{attribute 'linkalways'} 
{attribute 'no_explicit_call' := 'This FB is a CLASS and must be accessed using methods or properties'}
{attribute 'enable_dynamic_creation'}
FUNCTION_BLOCK Node_F_VN_CreateHighpassButterworthFilter EXTENDS VisionNode
VAR
    ipFilter : _ITcVnImage;
    nWidth : _UDINT(2);
    nHeight : _UDINT(2);
    bDoublePrecision : _BOOL(FALSE);
    bOriginAtCenter : _BOOL(FALSE);
    fCutoffDistance : _LREAL(1.0);
    nOrder : _UDINT(1);
    fScale : _LREAL(1.0);
    hrPrev : _HRESULT(S_OK);
	hresult : _HRESULT(S_OK);
END_VAR

METHOD PUBLIC  Clone : I_Node
VAR
	pNode : POINTER TO Node_F_VN_CreateHighpassButterworthFilter;
END_VAR
pNode := __NEW(Node_F_VN_CreateHighpassButterworthFilter);
Clone := pNode^;
END_METHOD

METHOD FB_init : BOOL
VAR_INPUT
	bInitRetains : BOOL; // if TRUE, the retain variables are initialized (warm start / cold start)
	bInCopyCode : BOOL;  // if TRUE, the instance afterwards gets moved into the copy code (online change)
END_VAR
AddParameter('nWidth', nWidth);
AddParameter('nHeight', nHeight);
AddParameter('bDoublePrecision', bDoublePrecision);
AddParameter('bOriginAtCenter', bOriginAtCenter);
AddParameter('fCutoffDistance', fCutoffDistance);
AddParameter('nOrder', nOrder);
AddParameter('fScale', fScale);
AddInput('hrPrev', hrPrev);
AddOutput('ipFilter', ipFilter);
AddOutput('hresult',hresult);
END_METHOD

METHOD PROTECTED OnExecute
hresult.Value := F_VN_CreateHighpassButterworthFilter(
    ipFilter := ipFilter.Value,
	nWidth := nWidth.Value,
    nHeight := nHeight.Value,
    bDoublePrecision := bDoublePrecision.Value,
    bOriginAtCenter := bOriginAtCenter.Value,
    fCutoffDistance := fCutoffDistance.Value,
    nOrder := nOrder.Value,
    fScale := fScale.Value,
	hrPrev:= hrPrev.Value);
END_METHOD

METHOD PUBLIC PreExecutionCheck
VAR_INPUT
	Check : I_PreExecutionChecks;
END_VAR
Check.IsTrue(nWidth.IsEven, 'nWidth must be an even number');
Check.IsTrue(nHeight.IsEven, 'nHeight must be an even number');
Check.IsTrue((nWidth.Value >= 2), 'nWidth must be greater than or equal to 2');
Check.IsTrue((nHeight.Value >= 2), 'nWidth must be greater than or equal to 2');
Check.IsTrue((fCutoffDistance.Value > 0), 'nCutoffDistance must be greater than 0');
Check.IsTrue((nOrder.Value > 0), 'nOrder must be greater than 0');
Check.IsTrue((fScale.Value > 0), 'fScale must be greater than 0');
END_METHOD

END_FUNCTION_BLOCK

(* stored: Version 1.1.0.1, ProductVersion 3.1.4024.13
   POU Node_F_VN_CreateHighpassButterworthFilter: Id {e6d8493b-b689-0c34-30ba-ecc7acc460ab}, SpecialFunc None
   Folder Constructor: Id {10b100ae-515d-058b-0a31-404109c7c72b}
   Method Clone: Id {01652cac-4fbc-0893-23d7-e4b31a061049}
   Method FB_init: Id {f6bc299e-12e4-0568-18ce-5851d752d7f8}
   Method OnExecute: Id {50d4bdba-af90-0a1e-0d48-b1fbc687bd5e}
   Method PreExecutionCheck: Id {3a822e6b-2830-092d-213d-515aa19a20b1} *)
